// TIA Portal V15.1 export
// export: Created 2020-06-12T07:35:52.6787109Z, ExportSetting None, DisplayName Totally Integrated Automation Portal, DisplayVersion V15.1, DisplayName TIA Portal Openness, DisplayVersion V15.1, DisplayName STEP 7 Professional, DisplayVersion V15.1, DisplayName STEP 7 Safety, DisplayVersion V15.1, DisplayName WinCC Advanced, DisplayVersion V15.1
FUNCTION "MELT_Setpoints" : Void   // FC90, FBD
{ S7_Optimized_Access := 'TRUE' }
// stored: SetENOAutomatically False
   VAR_TEMP
      tTmpU : Real;
      tPwrAdd : Real;
      tResAdd : Real;
      tCalcSW : Bool;
      tCalcMR : Bool;
      tCalcPwr : Bool;
      tCalcRes : Bool;
      tVar3 : Real;
      tHTPower : Real;
      tHTResistance : Real;
      tPmax : Real;
      tImax : Real;
      tUseST : Bool;
      tUseHT : Bool;
      tCosPhi : Real;
      tUlim : Real;
      tIlim : Real;
      tUseForOCT : Bool;
      tPset_ST : Real;
      tPset_OCT : Real;
   END_VAR
BEGIN

REGION Network 1: Clocks
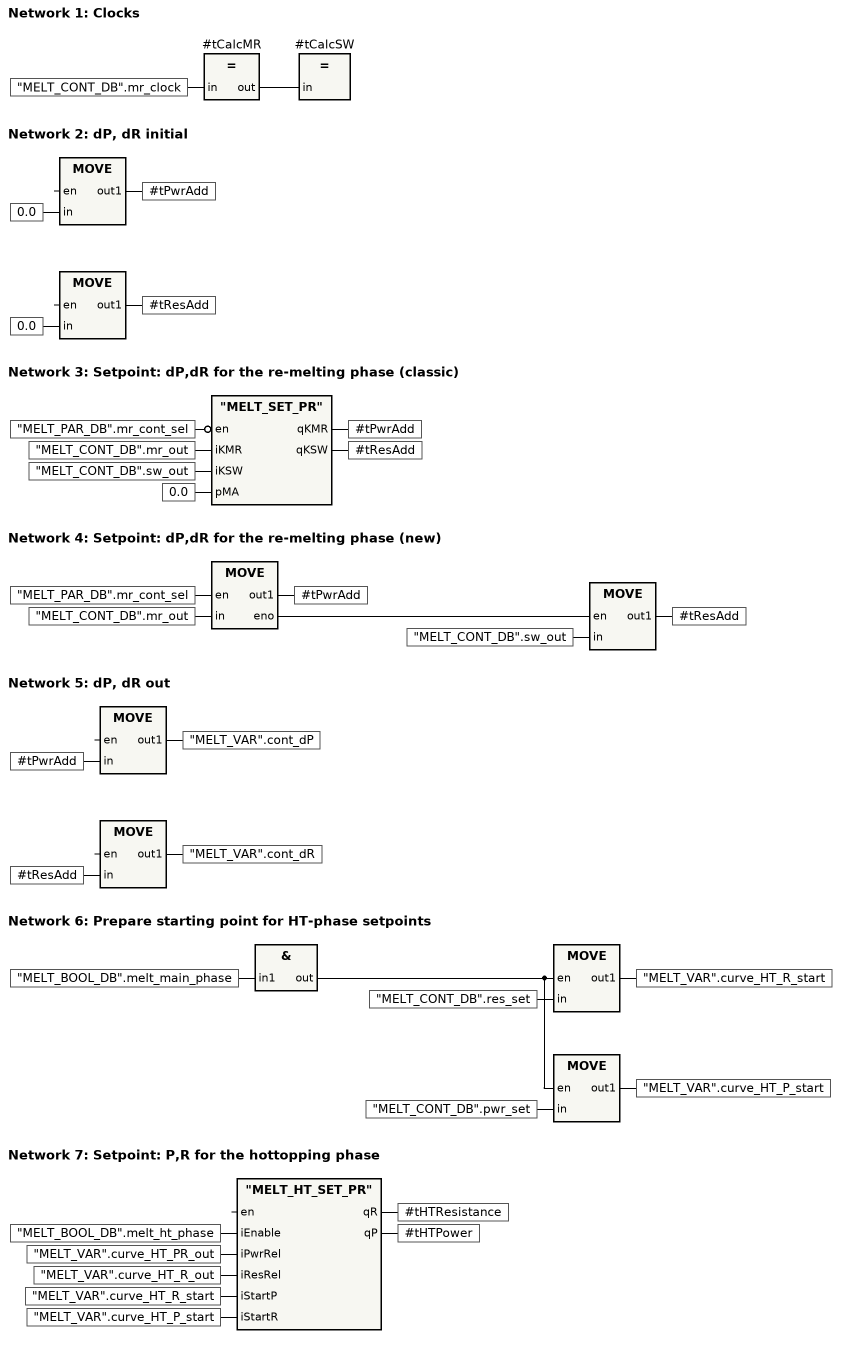
   #tCalcMR := "MELT_CONT_DB".mr_clock;
   #tCalcSW := "MELT_CONT_DB".mr_clock;
END_REGION

REGION Network 2: dP, dR initial
   #tPwrAdd := 0.0;
   #tResAdd := 0.0;
END_REGION

REGION Network 3: Setpoint: dP,dR for the re-melting phase (classic)
   IF NOT "MELT_PAR_DB".mr_cont_sel THEN
       "MELT_SET_PR"(iKMR := "MELT_CONT_DB".mr_out,
                     iKSW := "MELT_CONT_DB".sw_out,
                     pMA := 0.0,
                     qKMR => #tPwrAdd,
                     qKSW => #tResAdd);
   END_IF;
END_REGION

REGION Network 4: Setpoint: dP,dR for the re-melting phase (new)
   // If the MR-, Sw-controllers will configured for the physical units, we can use more simple calculation for P, R.
   // The output configuration for MR-cont can be power [kW], or a power changing [kW/min]
   // The output configuration for Sw-cont can be resistance [mOhm], or a resistance changing [mOhm/min]
   // 
   // A new bonus is smooth process regulation.
   IF "MELT_PAR_DB".mr_cont_sel THEN
       #tPwrAdd := "MELT_CONT_DB".mr_out;
       #tResAdd := "MELT_CONT_DB".sw_out;
   END_IF;
END_REGION

REGION Network 5: dP, dR out
   "MELT_VAR".cont_dP := #tPwrAdd;
   "MELT_VAR".cont_dR := #tResAdd;
END_REGION

REGION Network 6: Prepare starting point for HT-phase setpoints
   IF "MELT_BOOL_DB".melt_main_phase THEN
       "MELT_VAR".curve_HT_R_start := "MELT_CONT_DB".res_set;
       "MELT_VAR".curve_HT_P_start := "MELT_CONT_DB".pwr_set;
   END_IF;
END_REGION

REGION Network 7: Setpoint: P,R for the hottopping phase
   "MELT_HT_SET_PR"(iEnable := "MELT_BOOL_DB".melt_ht_phase,
                    iPwrRel := "MELT_VAR".curve_HT_PR_out,
                    iResRel := "MELT_VAR".curve_HT_R_out,
                    iStartP := "MELT_VAR".curve_HT_R_start,
                    iStartR := "MELT_VAR".curve_HT_P_start,
                    qR => #tHTResistance,
                    qP => #tHTPower);
END_REGION

REGION Network 8: Setpoint selectors flags
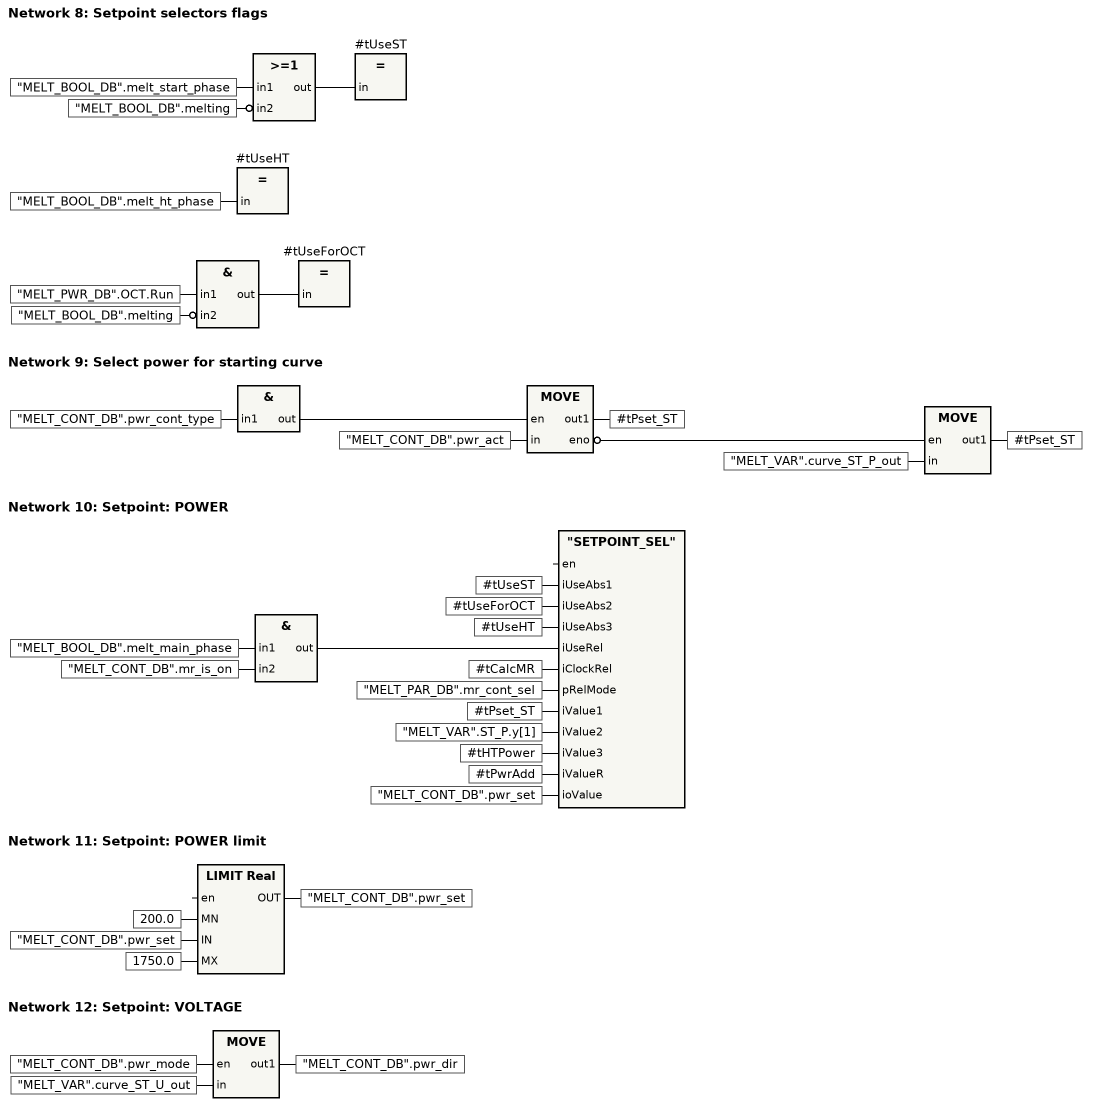
   #tUseST := "MELT_BOOL_DB".melt_start_phase OR NOT "MELT_BOOL_DB".melting;
   #tUseHT := "MELT_BOOL_DB".melt_ht_phase;
   #tUseForOCT := "MELT_PWR_DB".OCT.Run AND NOT "MELT_BOOL_DB".melting;
END_REGION

REGION Network 9: Select power for starting curve
   // NB A problem can happen if P_act = 0 (CB is OFF, electrode is out)
   IF "MELT_CONT_DB".pwr_cont_type THEN #tPset_ST := "MELT_CONT_DB".pwr_act; END_IF;
   IF NOT "MELT_CONT_DB".pwr_cont_type THEN #tPset_ST := "MELT_VAR".curve_ST_P_out; END_IF;
END_REGION

REGION Network 10: Setpoint: POWER
   "SETPOINT_SEL"(iUseAbs1 := #tUseST,
                  iUseAbs2 := #tUseForOCT,
                  iUseAbs3 := #tUseHT,
                  iUseRel := "MELT_BOOL_DB".melt_main_phase AND "MELT_CONT_DB".mr_is_on,
                  iClockRel := #tCalcMR,
                  pRelMode := "MELT_PAR_DB".mr_cont_sel,
                  iValue1 := #tPset_ST,
                  iValue2 := "MELT_VAR".ST_P.y[1],
                  iValue3 := #tHTPower,
                  iValueR := #tPwrAdd,
                  ioValue := "MELT_CONT_DB".pwr_set);
END_REGION

REGION Network 11: Setpoint: POWER limit
   // 2.000000e+002
   "MELT_CONT_DB".pwr_set := LIMIT(MN := 200.0, IN := "MELT_CONT_DB".pwr_set, MX := 1750.0);
END_REGION

REGION Network 12: Setpoint: VOLTAGE
   IF "MELT_CONT_DB".pwr_mode THEN "MELT_CONT_DB".pwr_dir := "MELT_VAR".curve_ST_U_out; END_IF;
END_REGION

REGION Network 13: Setpoint: RESISTANCE
   // During OCT the cos(phi) is always 1, and this fact does a voltage calculation wrong.
   // To avoid this we will use special seed for resistance R!
   // R! = Rmin / cos_phi^2
   // For this plant cos_phi = 0.2 and Rmin = 0.5 mOhm
   // R! = 0.5 / 0,04 = 12,5 mOhm
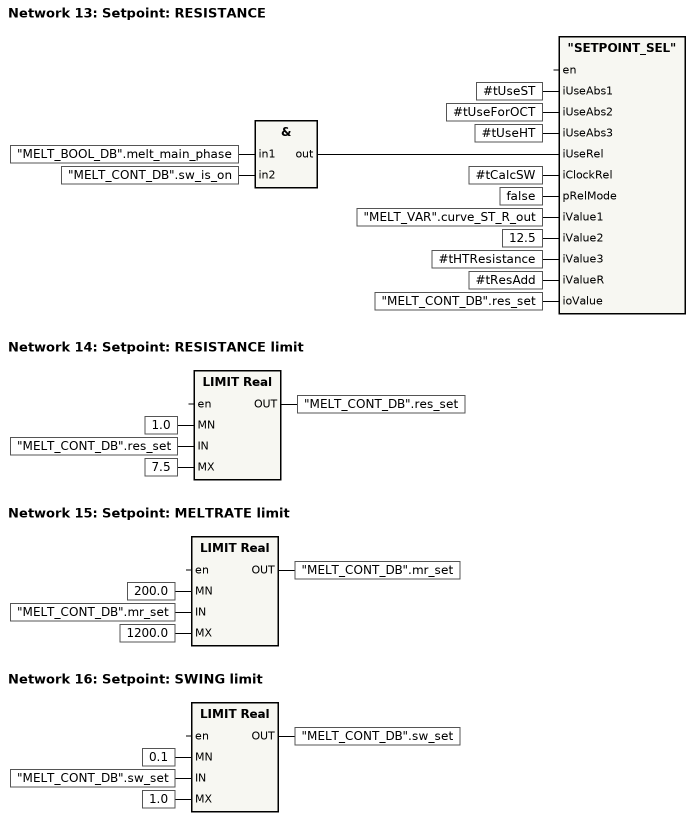
   "SETPOINT_SEL"(iUseAbs1 := #tUseST,
                  iUseAbs2 := #tUseForOCT,
                  iUseAbs3 := #tUseHT,
                  iUseRel := "MELT_BOOL_DB".melt_main_phase AND "MELT_CONT_DB".sw_is_on,
                  iClockRel := #tCalcSW,
                  pRelMode := false,
                  iValue1 := "MELT_VAR".curve_ST_R_out,
                  iValue2 := 12.5,
                  iValue3 := #tHTResistance,
                  iValueR := #tResAdd,
                  ioValue := "MELT_CONT_DB".res_set);
END_REGION

REGION Network 14: Setpoint: RESISTANCE limit
   // 2.000000e+002
   "MELT_CONT_DB".res_set := LIMIT(MN := 1.0, IN := "MELT_CONT_DB".res_set, MX := 7.5);
END_REGION

REGION Network 15: Setpoint: MELTRATE limit
   "MELT_CONT_DB".mr_set := LIMIT(MN := 200.0, IN := "MELT_CONT_DB".mr_set, MX := 1200.0);
END_REGION

REGION Network 16: Setpoint: SWING limit
   "MELT_CONT_DB".sw_set := LIMIT(MN := 0.1, IN := "MELT_CONT_DB".sw_set, MX := 1.0);
END_REGION
END_FUNCTION
